Staubli VAL3: isListEmpty.pgx

public program isListEmpty(bool& x_bEmpty[])
begin
  //-----------------------------------------------------------------------
  //Header begin
  //Description of program
  //  Test if the list of Items is empty.
  //
  //Input parameters
  //  bool x_bEmpty :
  //    role : Set to true if the list is empty and false otherwise
  //
  //Example
  //  call isListEmpty(l_bEmpty)
  //
  //History
  //  Creation : 28-04-08 - f.Rob
  //Header end
  //-----------------------------------------------------------------------
  if size(sItems)==1 and sItems[0]==""
    x_bEmpty=true
  else
    x_bEmpty=false
  endIf
end
